Staubli VAL3: refreshStatic.pgx

program refreshStatic()
  local string l_sMenu
  local num i
  local string l_sInstruction
  local num l_nSize
  local string l_sMessage
  local mdesc l_mDesc
  local num l_nTcpAction
  local string l_sName
  local string l_sEmpty
  local bool l_bStop
  local num l_nEmpty
  local num l_nIndexTool
  local TrajectoryItem l_tTraj
  local string l_sType
  local string l_sData
begin
  cls()
  //
  // set the view of the page..
  //
  // SET THE PAGE NUMBER
  use:nPage=100000
  // USE <>PROFILE for <>PAGE
  use:nPage=use:nPage+abs(limit(saveData:mode,0,2)-2)
  // load the menu page
  if saveData:language!="japanese"
    // SET THE VIEW OF THE PAGE
    call language:page(l_sMessage,use:nPage)
    // define the menu
    call use:stringToArray(l_sMessage,sMenu)
  else
    // japanese use the array for the menu
    call language:page(sMenu8,use:nPage)
    call use:stringCopy(sMenu8,sMenu)
  endIf
  //
  // polymorphism
  //
  // get the user Menu or special one
  call trajType:getFunctionEdit(sMenuUser)
  // OVERRIDE
  for i=0 to size(sMenuUser)-1
    if sMenuUser[i]!=""
      sMenu[i]=sMenuUser[i]
    endIf
  endFor
  // check for the here if not in cycle
  if cycleStatus:bCycle or cycleStatus:bSimulation
    sMenu[0]=""
  endIf
  // remove the insert delete in this page
  sMenu[5]=sMenu[6]=""
  if saveData:language!="japanese"
    // set the menu
    call use:setMenu(sMenu,true,3)
  else
    // set the menu
    call use:setMenu(sMenu,false,3)
  endIf
  call use:getMenu(sMenu,bButton)
  //
  // CREATE THE LIST
  //
  // define your list size for default
  // get the nSize
  call trajType:getSizeItem(false,l_nSize)
  call use:setSizeList(19,0,19,10)
  call use:setView(bLarge)
  // show the title...
  l_sName=sTrajName
  if !bLarge and len(sTrajName)>12
    // as japanese told us
    l_sName=left(sTrajName,9)+"¬"+right(sTrajName,2)
  endIf
  call use:listcreate(l_sName+" "+toString("3",nIndexItem+1)+"/"+toString("3",l_nSize))
  //
  call use:listadd(sList)
  //
  // refresh the cursor
  use:nView=nView
  // refresh the list
  call use:selectNewField(nSelected,nIndex,nView)
  // show the instruction
  l_sEmpty=""
  l_bStop=false
  l_nEmpty=0
  call trajType:getTrajItem(l_tTraj,nIndexItem)
  // select the action
  switch l_tTraj.nTcpAction
    case 1
      l_sInstruction="[ON],"
    break
    case 2
      l_sInstruction="[OFF],"
    break
    default
    break
  endSwitch
  l_sType=l_tTraj.iInstr[0].sType
  l_sData=l_tTraj.iInstr[0].sData
  call saveInOut:replaceIO(l_sData,l_sType,l_sData)
  l_sInstruction=l_sInstruction+l_sType+" "+l_sData
  for i=1 to size(l_tTraj.iInstr)-1
    if l_tTraj.iInstr[i].sType!=""
      l_sType=l_tTraj.iInstr[i].sType
      l_sData=l_tTraj.iInstr[i].sData
      call saveInOut:replaceIO(l_sData,l_sType,l_sData)
      l_sInstruction=l_sInstruction+","+l_sType+" "+l_sData
    endIf
  endFor
  call use:typeLen(0,12,l_sInstruction,40)
  // TOOL - FRAME
  if !bLarge
    call trajType:getTool(i)
    call language:message(l_sMessage,124)
    call tcp:getName(l_sName,i)
    call use:type(0,0,l_sMessage+":"+toString("",i)+" "+l_sName)
    call trajType:getFrameId(i)
    call language:message(l_sMessage,124)
    l_sName=saveData:fFrameItem[i].sName
    call use:type(0,1,"Frame:"+toString("",i)+" "+l_sName)
  endIf
end
